// TIA Portal V15.1 export
// export: Created 2024-05-17T05:38:57.1842107Z, ExportSetting WithDefaults, DisplayName Totally Integrated Automation Portal, DisplayVersion V15.1 Update 5, DisplayName TIA Portal Openness, DisplayVersion V15.1 Update 5, DisplayName SINAMICS Startdrive Advanced, DisplayVersion V15.1, DisplayName G130, G150, S120, S150, SINAMICS MV, S210, DisplayVersion V15.1, DisplayName G110M, G120, G120C, G120D, G120P, DisplayVersion V15.1, DisplayName STEP 7 Professional, DisplayVersion V15.1 Update 5, DisplayName STEP 7 Safety, DisplayVersion V15.1, DisplayName WinCC Professional, DisplayVersion V15.1 Update 5, DisplayName SIMATIC Visualization Architect, DisplayVersion V15.1
FUNCTION "209210ZS01Passiv" : Void   // FC323, FBD
TITLE = 209210ZS01Passiv
{ S7_Optimized_Access := 'FALSE' }
AUTHOR : VCC
NAME : LocFunc
VERSION : 0.1
// stored: AutoNumber false, IsIECCheckEnabled false, SetENOAutomatically False, UDAEnableTagReadback false
   VAR_OUTPUT
      O_AlarmA : Bool;   // Alarm A
      O_AlarmB : Bool;   // Alarm B
      O_AlarmC : Bool;   // Alarm C
      O_AlarmD : Bool;   // Alarm D
      O_AlarmABCondition : Bool;   // Alarms resetable
      H_IAnim : Word;   // Icon Animation
   END_VAR
   VAR_TEMP
      TEMP0 : Bool;
   END_VAR
BEGIN

REGION Network 1: **** --------------------- ET200sp I/O --------------------- ****
END_REGION

REGION Network 2: **** 2.2 - Alarms - Alarm Generation **** 209000AK03JX36QF5240 - ET200sp I/O - Safety Card QF5240
   // Passivation alarm - ET200sp I/O - Safety Card QF5240
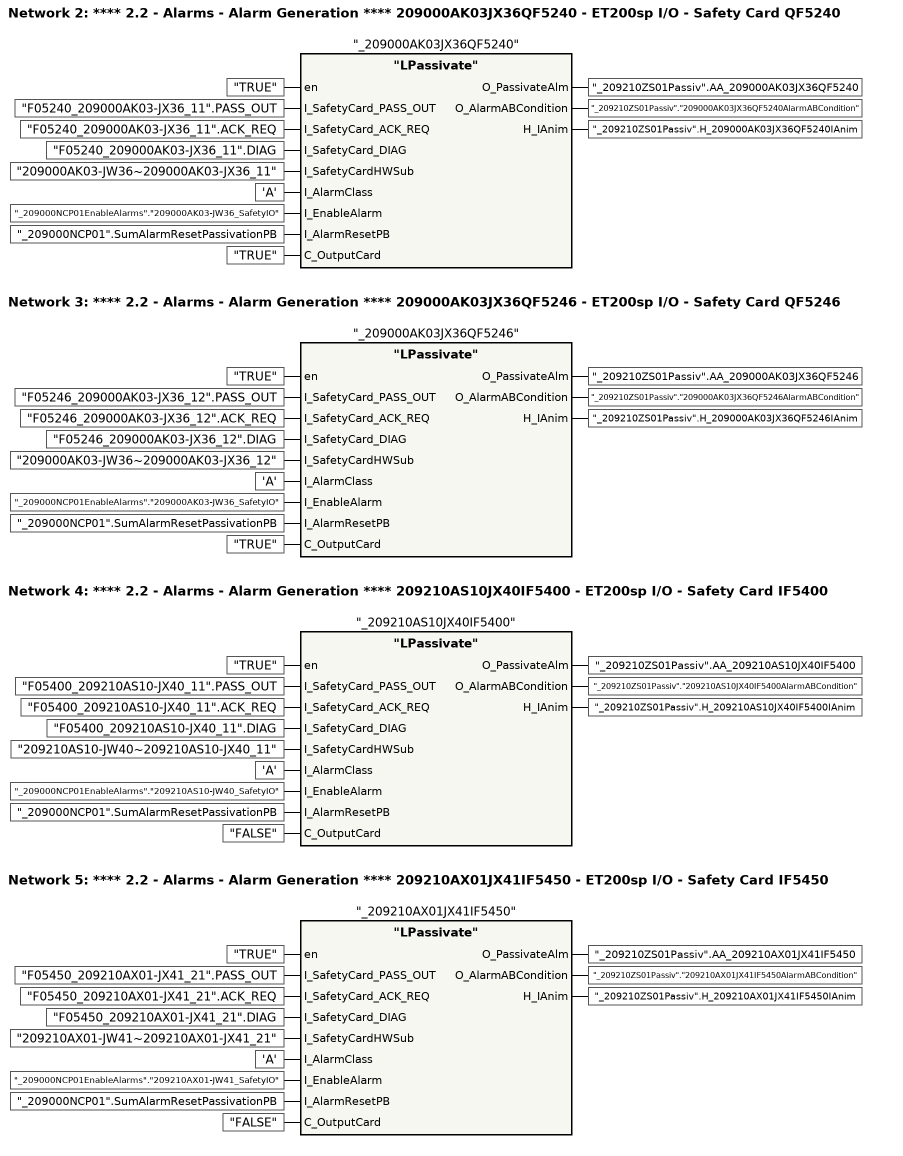
   IF "TRUE" THEN
       "_209000AK03JX36QF5240"(I_SafetyCard_PASS_OUT := "F05240_209000AK03-JX36_11".PASS_OUT,   // "LPassivate"
                               I_SafetyCard_ACK_REQ := "F05240_209000AK03-JX36_11".ACK_REQ,
                               I_SafetyCard_DIAG := "F05240_209000AK03-JX36_11".DIAG,
                               I_SafetyCardHWSub := "209000AK03-JW36~209000AK03-JX36_11",
                               I_AlarmClass := 'A',
                               I_EnableAlarm := "_209000NCP01EnableAlarms"."209000AK03-JW36_SafetyIO",
                               I_AlarmResetPB := "_209000NCP01".SumAlarmResetPassivationPB,
                               C_OutputCard := "TRUE",
                               O_PassivateAlm => "_209210ZS01Passiv".AA_209000AK03JX36QF5240,
                               O_AlarmABCondition => "_209210ZS01Passiv"."209000AK03JX36QF5240AlarmABCondition",
                               H_IAnim => "_209210ZS01Passiv".H_209000AK03JX36QF5240IAnim);
   END_IF;
END_REGION

REGION Network 3: **** 2.2 - Alarms - Alarm Generation **** 209000AK03JX36QF5246 - ET200sp I/O - Safety Card QF5246
   // Passivation alarm - ET200sp I/O - Safety Card QF5246
   IF "TRUE" THEN
       "_209000AK03JX36QF5246"(I_SafetyCard_PASS_OUT := "F05246_209000AK03-JX36_12".PASS_OUT,   // "LPassivate"
                               I_SafetyCard_ACK_REQ := "F05246_209000AK03-JX36_12".ACK_REQ,
                               I_SafetyCard_DIAG := "F05246_209000AK03-JX36_12".DIAG,
                               I_SafetyCardHWSub := "209000AK03-JW36~209000AK03-JX36_12",
                               I_AlarmClass := 'A',
                               I_EnableAlarm := "_209000NCP01EnableAlarms"."209000AK03-JW36_SafetyIO",
                               I_AlarmResetPB := "_209000NCP01".SumAlarmResetPassivationPB,
                               C_OutputCard := "TRUE",
                               O_PassivateAlm => "_209210ZS01Passiv".AA_209000AK03JX36QF5246,
                               O_AlarmABCondition => "_209210ZS01Passiv"."209000AK03JX36QF5246AlarmABCondition",
                               H_IAnim => "_209210ZS01Passiv".H_209000AK03JX36QF5246IAnim);
   END_IF;
END_REGION

REGION Network 4: **** 2.2 - Alarms - Alarm Generation **** 209210AS10JX40IF5400 - ET200sp I/O - Safety Card IF5400
   // Passivation alarm - ET200sp I/O - Safety Card IF5400
   IF "TRUE" THEN
       "_209210AS10JX40IF5400"(I_SafetyCard_PASS_OUT := "F05400_209210AS10-JX40_11".PASS_OUT,   // "LPassivate"
                               I_SafetyCard_ACK_REQ := "F05400_209210AS10-JX40_11".ACK_REQ,
                               I_SafetyCard_DIAG := "F05400_209210AS10-JX40_11".DIAG,
                               I_SafetyCardHWSub := "209210AS10-JW40~209210AS10-JX40_11",
                               I_AlarmClass := 'A',
                               I_EnableAlarm := "_209000NCP01EnableAlarms"."209210AS10-JW40_SafetyIO",
                               I_AlarmResetPB := "_209000NCP01".SumAlarmResetPassivationPB,
                               C_OutputCard := "FALSE",
                               O_PassivateAlm => "_209210ZS01Passiv".AA_209210AS10JX40IF5400,
                               O_AlarmABCondition => "_209210ZS01Passiv"."209210AS10JX40IF5400AlarmABCondition",
                               H_IAnim => "_209210ZS01Passiv".H_209210AS10JX40IF5400IAnim);
   END_IF;
END_REGION

REGION Network 5: **** 2.2 - Alarms - Alarm Generation **** 209210AX01JX41IF5450 - ET200sp I/O - Safety Card IF5450
   // Passivation alarm - ET200sp I/O - Safety Card IF5450
   IF "TRUE" THEN
       "_209210AX01JX41IF5450"(I_SafetyCard_PASS_OUT := "F05450_209210AX01-JX41_21".PASS_OUT,   // "LPassivate"
                               I_SafetyCard_ACK_REQ := "F05450_209210AX01-JX41_21".ACK_REQ,
                               I_SafetyCard_DIAG := "F05450_209210AX01-JX41_21".DIAG,
                               I_SafetyCardHWSub := "209210AX01-JW41~209210AX01-JX41_21",
                               I_AlarmClass := 'A',
                               I_EnableAlarm := "_209000NCP01EnableAlarms"."209210AX01-JW41_SafetyIO",
                               I_AlarmResetPB := "_209000NCP01".SumAlarmResetPassivationPB,
                               C_OutputCard := "FALSE",
                               O_PassivateAlm => "_209210ZS01Passiv".AA_209210AX01JX41IF5450,
                               O_AlarmABCondition => "_209210ZS01Passiv"."209210AX01JX41IF5450AlarmABCondition",
                               H_IAnim => "_209210ZS01Passiv".H_209210AX01JX41IF5450IAnim);
   END_IF;
END_REGION

REGION Network 6: **** 2.2 - Alarms - Alarm Generation **** 209210AS11JX42IF5500 - ET200sp I/O - Safety Card IF5500
   // Passivation alarm - ET200sp I/O - Safety Card IF5500
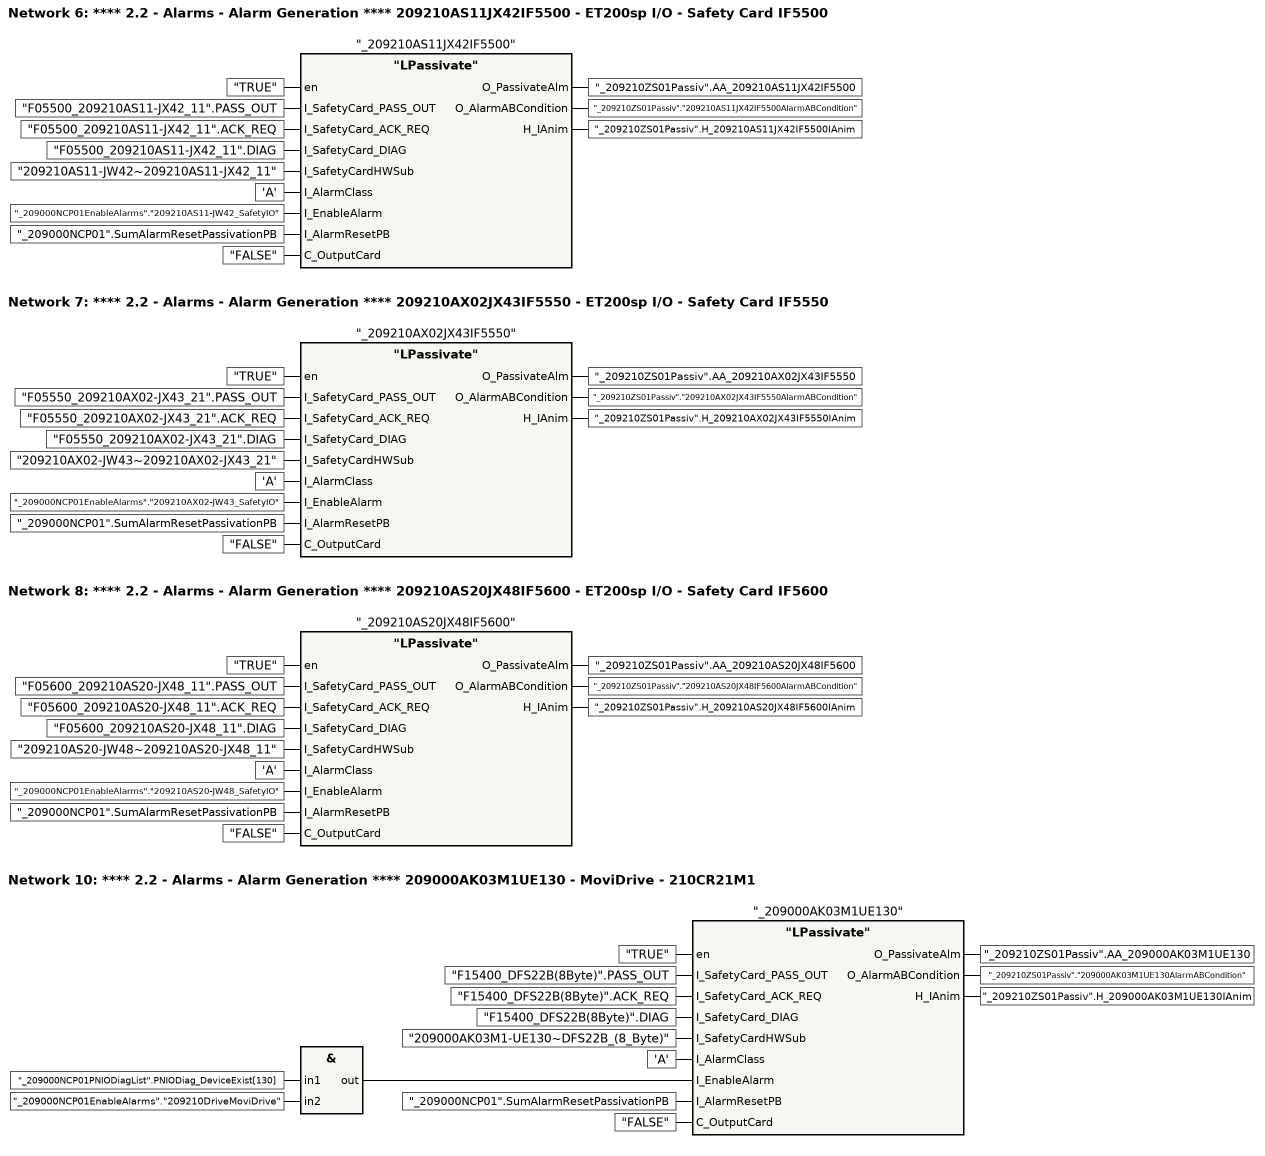
   IF "TRUE" THEN
       "_209210AS11JX42IF5500"(I_SafetyCard_PASS_OUT := "F05500_209210AS11-JX42_11".PASS_OUT,   // "LPassivate"
                               I_SafetyCard_ACK_REQ := "F05500_209210AS11-JX42_11".ACK_REQ,
                               I_SafetyCard_DIAG := "F05500_209210AS11-JX42_11".DIAG,
                               I_SafetyCardHWSub := "209210AS11-JW42~209210AS11-JX42_11",
                               I_AlarmClass := 'A',
                               I_EnableAlarm := "_209000NCP01EnableAlarms"."209210AS11-JW42_SafetyIO",
                               I_AlarmResetPB := "_209000NCP01".SumAlarmResetPassivationPB,
                               C_OutputCard := "FALSE",
                               O_PassivateAlm => "_209210ZS01Passiv".AA_209210AS11JX42IF5500,
                               O_AlarmABCondition => "_209210ZS01Passiv"."209210AS11JX42IF5500AlarmABCondition",
                               H_IAnim => "_209210ZS01Passiv".H_209210AS11JX42IF5500IAnim);
   END_IF;
END_REGION

REGION Network 7: **** 2.2 - Alarms - Alarm Generation **** 209210AX02JX43IF5550 - ET200sp I/O - Safety Card IF5550
   // Passivation alarm - ET200sp I/O - Safety Card IF5550
   IF "TRUE" THEN
       "_209210AX02JX43IF5550"(I_SafetyCard_PASS_OUT := "F05550_209210AX02-JX43_21".PASS_OUT,   // "LPassivate"
                               I_SafetyCard_ACK_REQ := "F05550_209210AX02-JX43_21".ACK_REQ,
                               I_SafetyCard_DIAG := "F05550_209210AX02-JX43_21".DIAG,
                               I_SafetyCardHWSub := "209210AX02-JW43~209210AX02-JX43_21",
                               I_AlarmClass := 'A',
                               I_EnableAlarm := "_209000NCP01EnableAlarms"."209210AX02-JW43_SafetyIO",
                               I_AlarmResetPB := "_209000NCP01".SumAlarmResetPassivationPB,
                               C_OutputCard := "FALSE",
                               O_PassivateAlm => "_209210ZS01Passiv".AA_209210AX02JX43IF5550,
                               O_AlarmABCondition => "_209210ZS01Passiv"."209210AX02JX43IF5550AlarmABCondition",
                               H_IAnim => "_209210ZS01Passiv".H_209210AX02JX43IF5550IAnim);
   END_IF;
END_REGION

REGION Network 8: **** 2.2 - Alarms - Alarm Generation **** 209210AS20JX48IF5600 - ET200sp I/O - Safety Card IF5600
   // Passivation alarm - ET200sp I/O - Safety Card IF5600
   IF "TRUE" THEN
       "_209210AS20JX48IF5600"(I_SafetyCard_PASS_OUT := "F05600_209210AS20-JX48_11".PASS_OUT,   // "LPassivate"
                               I_SafetyCard_ACK_REQ := "F05600_209210AS20-JX48_11".ACK_REQ,
                               I_SafetyCard_DIAG := "F05600_209210AS20-JX48_11".DIAG,
                               I_SafetyCardHWSub := "209210AS20-JW48~209210AS20-JX48_11",
                               I_AlarmClass := 'A',
                               I_EnableAlarm := "_209000NCP01EnableAlarms"."209210AS20-JW48_SafetyIO",
                               I_AlarmResetPB := "_209000NCP01".SumAlarmResetPassivationPB,
                               C_OutputCard := "FALSE",
                               O_PassivateAlm => "_209210ZS01Passiv".AA_209210AS20JX48IF5600,
                               O_AlarmABCondition => "_209210ZS01Passiv"."209210AS20JX48IF5600AlarmABCondition",
                               H_IAnim => "_209210ZS01Passiv".H_209210AS20JX48IF5600IAnim);
   END_IF;
END_REGION

REGION Network 9: **** --------------------- Drive --------------------- ****
END_REGION

REGION Network 10: **** 2.2 - Alarms - Alarm Generation **** 209000AK03M1UE130 - MoviDrive - 210CR21M1
   // Passivation alarm - MoviDrive - 210CR21M1
   IF "TRUE" THEN
       "_209000AK03M1UE130"(I_SafetyCard_PASS_OUT := "F15400_DFS22B(8Byte)".PASS_OUT,   // "LPassivate"
                            I_SafetyCard_ACK_REQ := "F15400_DFS22B(8Byte)".ACK_REQ,
                            I_SafetyCard_DIAG := "F15400_DFS22B(8Byte)".DIAG,
                            I_SafetyCardHWSub := "209000AK03M1-UE130~DFS22B_(8_Byte)",
                            I_AlarmClass := 'A',
                            I_EnableAlarm := "_209000NCP01PNIODiagList".PNIODiag_DeviceExist[130] AND "_209000NCP01EnableAlarms"."209210DriveMoviDrive",
                            I_AlarmResetPB := "_209000NCP01".SumAlarmResetPassivationPB,
                            C_OutputCard := "FALSE",
                            O_PassivateAlm => "_209210ZS01Passiv".AA_209000AK03M1UE130,
                            O_AlarmABCondition => "_209210ZS01Passiv"."209000AK03M1UE130AlarmABCondition",
                            H_IAnim => "_209210ZS01Passiv".H_209000AK03M1UE130IAnim);
   END_IF;
END_REGION

REGION Network 11: **** 2.2 - Alarms - Alarm Generation **** 209000AK03M4UE131 - MoviDrive - 210CS22M4ME1 (Power)
   // Passivation alarm - MoviDrive - 210CS22M4ME1 (Power)
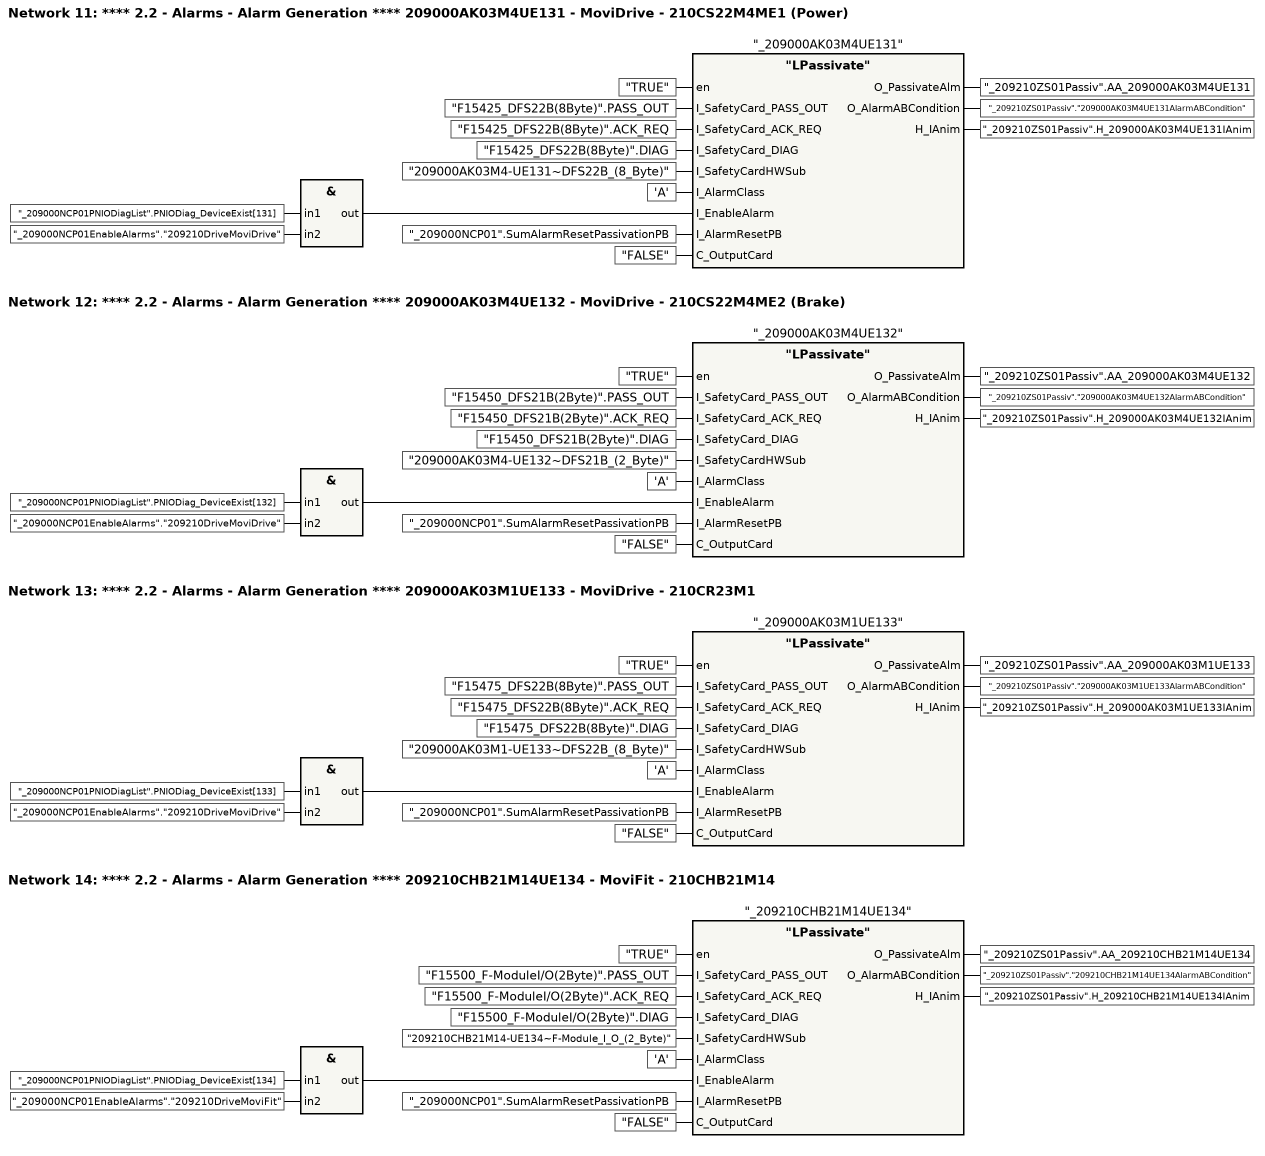
   IF "TRUE" THEN
       "_209000AK03M4UE131"(I_SafetyCard_PASS_OUT := "F15425_DFS22B(8Byte)".PASS_OUT,   // "LPassivate"
                            I_SafetyCard_ACK_REQ := "F15425_DFS22B(8Byte)".ACK_REQ,
                            I_SafetyCard_DIAG := "F15425_DFS22B(8Byte)".DIAG,
                            I_SafetyCardHWSub := "209000AK03M4-UE131~DFS22B_(8_Byte)",
                            I_AlarmClass := 'A',
                            I_EnableAlarm := "_209000NCP01PNIODiagList".PNIODiag_DeviceExist[131] AND "_209000NCP01EnableAlarms"."209210DriveMoviDrive",
                            I_AlarmResetPB := "_209000NCP01".SumAlarmResetPassivationPB,
                            C_OutputCard := "FALSE",
                            O_PassivateAlm => "_209210ZS01Passiv".AA_209000AK03M4UE131,
                            O_AlarmABCondition => "_209210ZS01Passiv"."209000AK03M4UE131AlarmABCondition",
                            H_IAnim => "_209210ZS01Passiv".H_209000AK03M4UE131IAnim);
   END_IF;
END_REGION

REGION Network 12: **** 2.2 - Alarms - Alarm Generation **** 209000AK03M4UE132 - MoviDrive - 210CS22M4ME2 (Brake)
   // Passivation alarm - MoviDrive - 210CS22M4ME2 (Brake)
   IF "TRUE" THEN
       "_209000AK03M4UE132"(I_SafetyCard_PASS_OUT := "F15450_DFS21B(2Byte)".PASS_OUT,   // "LPassivate"
                            I_SafetyCard_ACK_REQ := "F15450_DFS21B(2Byte)".ACK_REQ,
                            I_SafetyCard_DIAG := "F15450_DFS21B(2Byte)".DIAG,
                            I_SafetyCardHWSub := "209000AK03M4-UE132~DFS21B_(2_Byte)",
                            I_AlarmClass := 'A',
                            I_EnableAlarm := "_209000NCP01PNIODiagList".PNIODiag_DeviceExist[132] AND "_209000NCP01EnableAlarms"."209210DriveMoviDrive",
                            I_AlarmResetPB := "_209000NCP01".SumAlarmResetPassivationPB,
                            C_OutputCard := "FALSE",
                            O_PassivateAlm => "_209210ZS01Passiv".AA_209000AK03M4UE132,
                            O_AlarmABCondition => "_209210ZS01Passiv"."209000AK03M4UE132AlarmABCondition",
                            H_IAnim => "_209210ZS01Passiv".H_209000AK03M4UE132IAnim);
   END_IF;
END_REGION

REGION Network 13: **** 2.2 - Alarms - Alarm Generation **** 209000AK03M1UE133 - MoviDrive - 210CR23M1
   // Passivation alarm - MoviDrive - 210CR23M1
   IF "TRUE" THEN
       "_209000AK03M1UE133"(I_SafetyCard_PASS_OUT := "F15475_DFS22B(8Byte)".PASS_OUT,   // "LPassivate"
                            I_SafetyCard_ACK_REQ := "F15475_DFS22B(8Byte)".ACK_REQ,
                            I_SafetyCard_DIAG := "F15475_DFS22B(8Byte)".DIAG,
                            I_SafetyCardHWSub := "209000AK03M1-UE133~DFS22B_(8_Byte)",
                            I_AlarmClass := 'A',
                            I_EnableAlarm := "_209000NCP01PNIODiagList".PNIODiag_DeviceExist[133] AND "_209000NCP01EnableAlarms"."209210DriveMoviDrive",
                            I_AlarmResetPB := "_209000NCP01".SumAlarmResetPassivationPB,
                            C_OutputCard := "FALSE",
                            O_PassivateAlm => "_209210ZS01Passiv".AA_209000AK03M1UE133,
                            O_AlarmABCondition => "_209210ZS01Passiv"."209000AK03M1UE133AlarmABCondition",
                            H_IAnim => "_209210ZS01Passiv".H_209000AK03M1UE133IAnim);
   END_IF;
END_REGION

REGION Network 14: **** 2.2 - Alarms - Alarm Generation **** 209210CHB21M14UE134 - MoviFit - 210CHB21M14
   // Passivation alarm - MoviFit - 210CHB21M14
   IF "TRUE" THEN
       "_209210CHB21M14UE134"(I_SafetyCard_PASS_OUT := "F15500_F-ModuleI/O(2Byte)".PASS_OUT,   // "LPassivate"
                              I_SafetyCard_ACK_REQ := "F15500_F-ModuleI/O(2Byte)".ACK_REQ,
                              I_SafetyCard_DIAG := "F15500_F-ModuleI/O(2Byte)".DIAG,
                              I_SafetyCardHWSub := "209210CHB21M14-UE134~F-Module_I_O_(2_Byte)",
                              I_AlarmClass := 'A',
                              I_EnableAlarm := "_209000NCP01PNIODiagList".PNIODiag_DeviceExist[134] AND "_209000NCP01EnableAlarms"."209210DriveMoviFit",
                              I_AlarmResetPB := "_209000NCP01".SumAlarmResetPassivationPB,
                              C_OutputCard := "FALSE",
                              O_PassivateAlm => "_209210ZS01Passiv".AA_209210CHB21M14UE134,
                              O_AlarmABCondition => "_209210ZS01Passiv"."209210CHB21M14UE134AlarmABCondition",
                              H_IAnim => "_209210ZS01Passiv".H_209210CHB21M14UE134IAnim);
   END_IF;
END_REGION

REGION Network 15: **** -------------------------------------------------- ****
END_REGION

REGION Network 16: **** 4.6 - Machine Status - Indications **** Icon animation
   // Icon animation
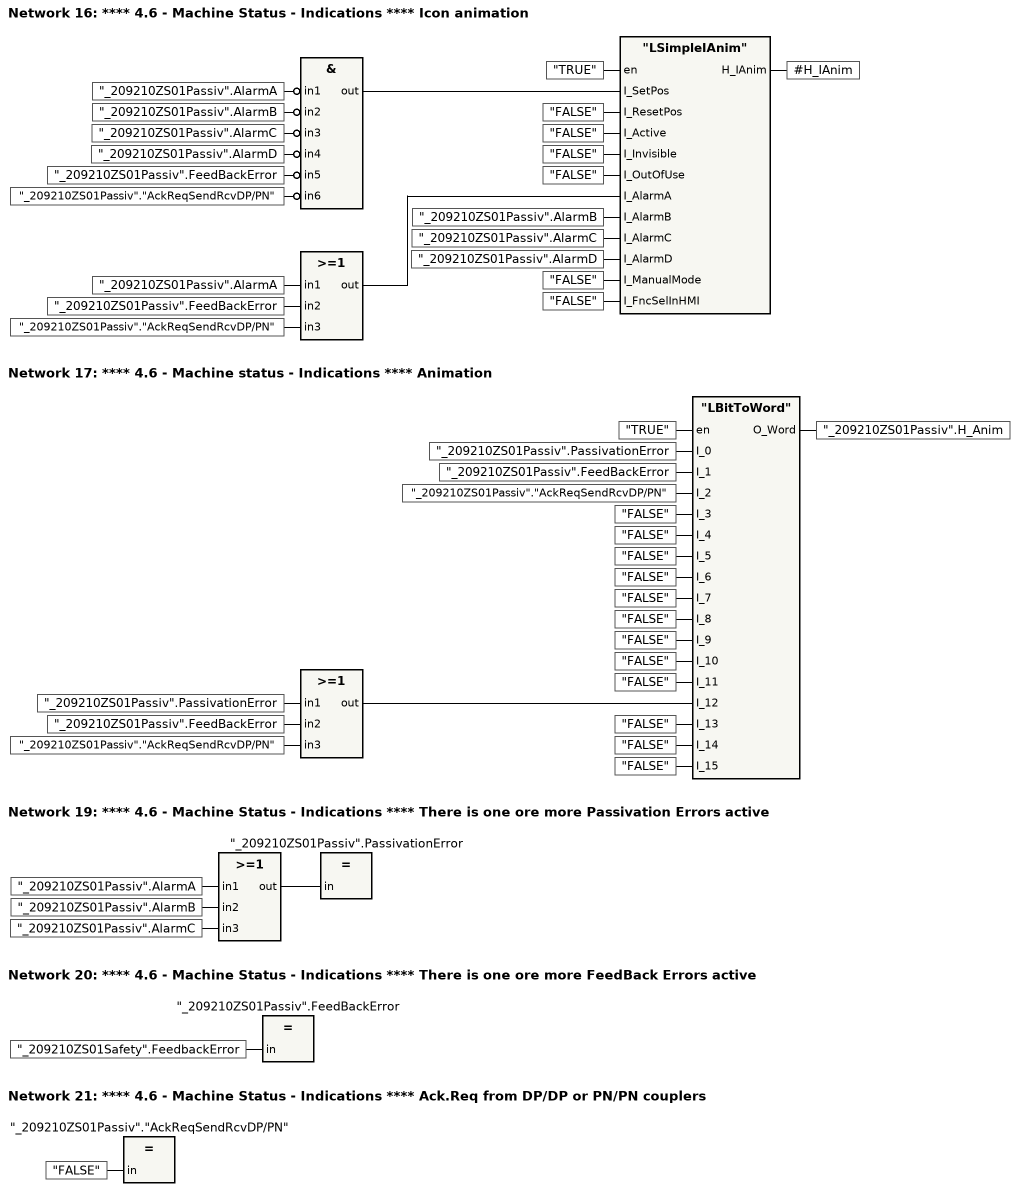
   IF "TRUE" THEN
       "LSimpleIAnim"(I_SetPos := NOT "_209210ZS01Passiv".AlarmA AND NOT "_209210ZS01Passiv".AlarmB AND NOT "_209210ZS01Passiv".AlarmC AND NOT "_209210ZS01Passiv".AlarmD AND NOT "_209210ZS01Passiv".FeedBackError AND NOT "_209210ZS01Passiv"."AckReqSendRcvDP/PN",
                      I_ResetPos := "FALSE",
                      I_Active := "FALSE",
                      I_Invisible := "FALSE",
                      I_OutOfUse := "FALSE",
                      I_AlarmA := "_209210ZS01Passiv".AlarmA OR "_209210ZS01Passiv".FeedBackError OR "_209210ZS01Passiv"."AckReqSendRcvDP/PN",
                      I_AlarmB := "_209210ZS01Passiv".AlarmB,
                      I_AlarmC := "_209210ZS01Passiv".AlarmC,
                      I_AlarmD := "_209210ZS01Passiv".AlarmD,
                      I_ManualMode := "FALSE",
                      I_FncSelInHMI := "FALSE",
                      H_IAnim => #H_IAnim);
   END_IF;
END_REGION

REGION Network 17: **** 4.6 - Machine status - Indications **** Animation
   // Animation
   IF "TRUE" THEN
       "LBitToWord"(I_0 := "_209210ZS01Passiv".PassivationError,
                    I_1 := "_209210ZS01Passiv".FeedBackError,
                    I_2 := "_209210ZS01Passiv"."AckReqSendRcvDP/PN",
                    I_3 := "FALSE",
                    I_4 := "FALSE",
                    I_5 := "FALSE",
                    I_6 := "FALSE",
                    I_7 := "FALSE",
                    I_8 := "FALSE",
                    I_9 := "FALSE",
                    I_10 := "FALSE",
                    I_11 := "FALSE",
                    I_12 := "_209210ZS01Passiv".PassivationError OR "_209210ZS01Passiv".FeedBackError OR "_209210ZS01Passiv"."AckReqSendRcvDP/PN",
                    I_13 := "FALSE",
                    I_14 := "FALSE",
                    I_15 := "FALSE",
                    O_Word => "_209210ZS01Passiv".H_Anim);
   END_IF;
END_REGION

NETWORK
TITLE = **** 4.6 - Machine Status - Indications **** Animation DB number
// DB number
      OPN   "_209210ZS01Passiv";
      L     DBNO;
      T     "_209210ZS01Passiv".H_DBnr;

REGION Network 19: **** 4.6 - Machine Status - Indications **** There is one ore more Passivation Errors active
   // There is one ore more Passivation Errors active
   "_209210ZS01Passiv".PassivationError := "_209210ZS01Passiv".AlarmA OR "_209210ZS01Passiv".AlarmB OR "_209210ZS01Passiv".AlarmC;
END_REGION

REGION Network 20: **** 4.6 - Machine Status - Indications **** There is one ore more FeedBack Errors active
   // There is one ore more FeedBack Errors active
   "_209210ZS01Passiv".FeedBackError := "_209210ZS01Safety".FeedbackError;
END_REGION

REGION Network 21: **** 4.6 - Machine Status - Indications **** Ack.Req from DP/DP or PN/PN couplers
   // Ack.Req from DP/DP or PN/PN couplers
   "_209210ZS01Passiv"."AckReqSendRcvDP/PN" := "FALSE";
END_REGION

REGION Network 22: **** 9 - Alarm Summary **** Alarm AB Condition
   // Alarm AB condition
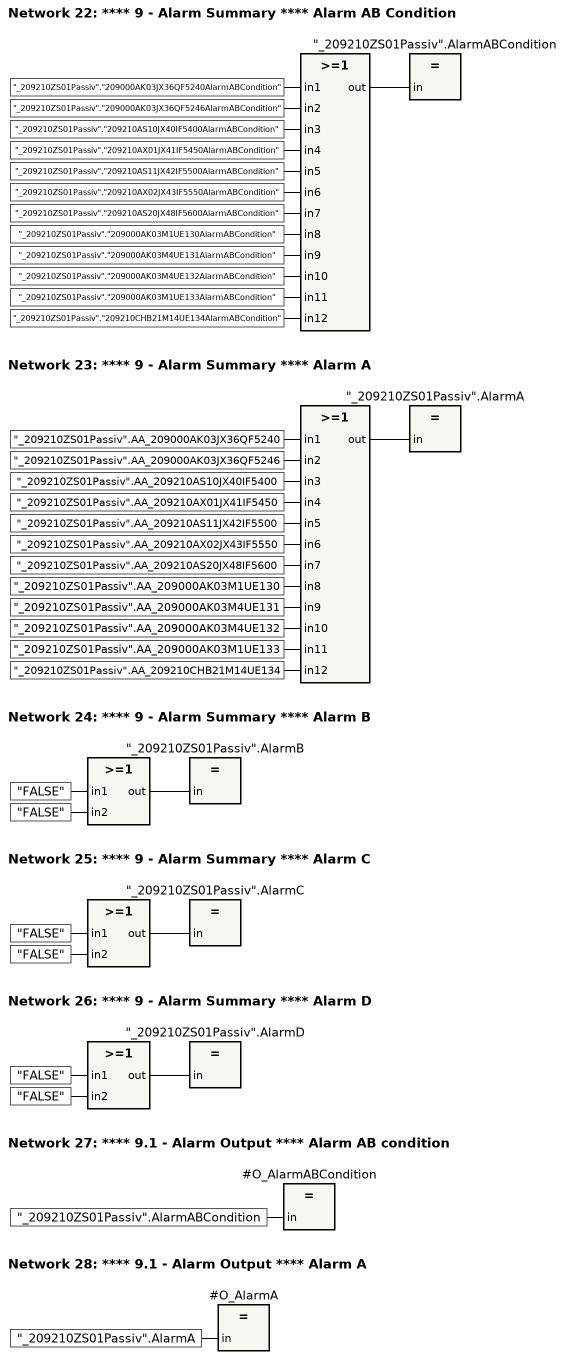
   "_209210ZS01Passiv".AlarmABCondition := "_209210ZS01Passiv"."209000AK03JX36QF5240AlarmABCondition" OR "_209210ZS01Passiv"."209000AK03JX36QF5246AlarmABCondition" OR "_209210ZS01Passiv"."209210AS10JX40IF5400AlarmABCondition" OR "_209210ZS01Passiv"."209210AX01JX41IF5450AlarmABCondition" OR "_209210ZS01Passiv"."209210AS11JX42IF5500AlarmABCondition" OR "_209210ZS01Passiv"."209210AX02JX43IF5550AlarmABCondition" OR "_209210ZS01Passiv"."209210AS20JX48IF5600AlarmABCondition" OR "_209210ZS01Passiv"."209000AK03M1UE130AlarmABCondition" OR "_209210ZS01Passiv"."209000AK03M4UE131AlarmABCondition" OR "_209210ZS01Passiv"."209000AK03M4UE132AlarmABCondition" OR "_209210ZS01Passiv"."209000AK03M1UE133AlarmABCondition" OR "_209210ZS01Passiv"."209210CHB21M14UE134AlarmABCondition";
END_REGION

REGION Network 23: **** 9 - Alarm Summary **** Alarm A
   // Summary of alarms A
   "_209210ZS01Passiv".AlarmA := "_209210ZS01Passiv".AA_209000AK03JX36QF5240 OR "_209210ZS01Passiv".AA_209000AK03JX36QF5246 OR "_209210ZS01Passiv".AA_209210AS10JX40IF5400 OR "_209210ZS01Passiv".AA_209210AX01JX41IF5450 OR "_209210ZS01Passiv".AA_209210AS11JX42IF5500 OR "_209210ZS01Passiv".AA_209210AX02JX43IF5550 OR "_209210ZS01Passiv".AA_209210AS20JX48IF5600 OR "_209210ZS01Passiv".AA_209000AK03M1UE130 OR "_209210ZS01Passiv".AA_209000AK03M4UE131 OR "_209210ZS01Passiv".AA_209000AK03M4UE132 OR "_209210ZS01Passiv".AA_209000AK03M1UE133 OR "_209210ZS01Passiv".AA_209210CHB21M14UE134;
END_REGION

REGION Network 24: **** 9 - Alarm Summary **** Alarm B
   // Summary of alarms B
   "_209210ZS01Passiv".AlarmB := "FALSE" OR "FALSE";
END_REGION

REGION Network 25: **** 9 - Alarm Summary **** Alarm C
   // Summary of alarms C
   "_209210ZS01Passiv".AlarmC := "FALSE" OR "FALSE";
END_REGION

REGION Network 26: **** 9 - Alarm Summary **** Alarm D
   // Summary of alarms D
   "_209210ZS01Passiv".AlarmD := "FALSE" OR "FALSE";
END_REGION

REGION Network 27: **** 9.1 - Alarm Output **** Alarm AB condition
   // Alarm AB condition
   #O_AlarmABCondition := "_209210ZS01Passiv".AlarmABCondition;
END_REGION

REGION Network 28: **** 9.1 - Alarm Output **** Alarm A
   // Output Alarm A
   #O_AlarmA := "_209210ZS01Passiv".AlarmA;
END_REGION

REGION Network 29: **** 9.1 - Alarm Output **** Alarm B
   // Output Alarm B
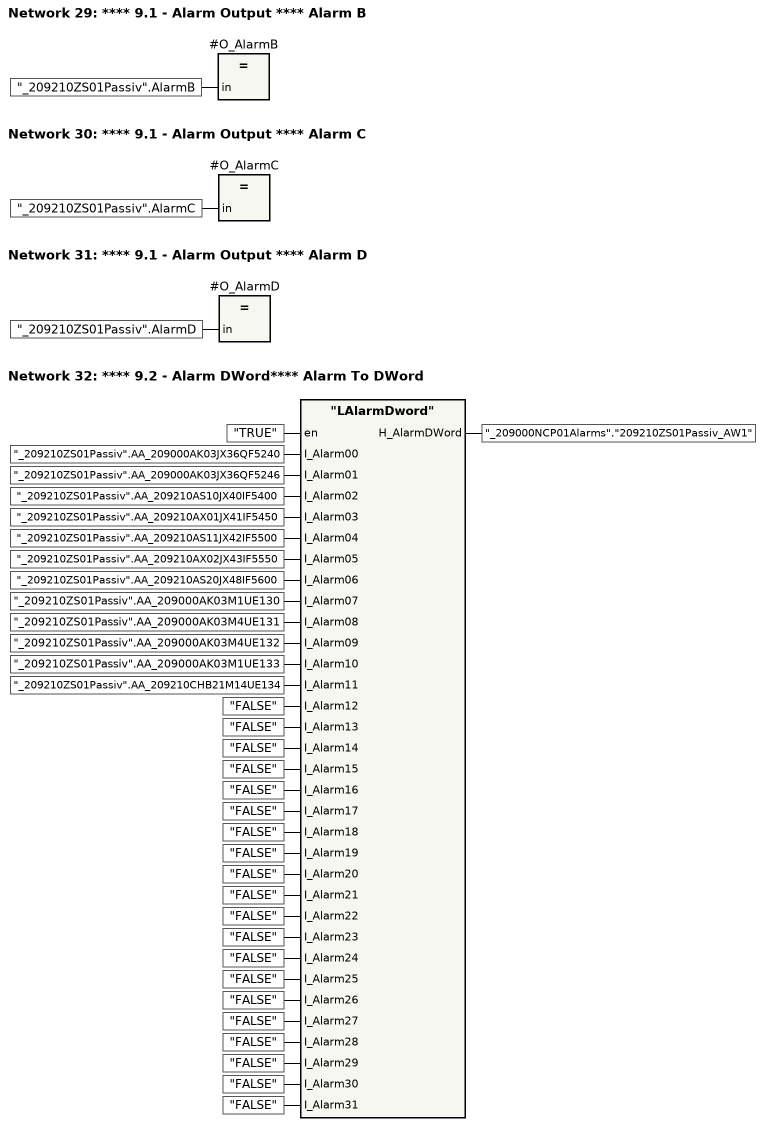
   #O_AlarmB := "_209210ZS01Passiv".AlarmB;
END_REGION

REGION Network 30: **** 9.1 - Alarm Output **** Alarm C
   // Output Alarm C
   #O_AlarmC := "_209210ZS01Passiv".AlarmC;
END_REGION

REGION Network 31: **** 9.1 - Alarm Output **** Alarm D
   // Output Alarm D
   #O_AlarmD := "_209210ZS01Passiv".AlarmD;
END_REGION

REGION Network 32: **** 9.2 - Alarm DWord**** Alarm To DWord
   // Alarm Word
   IF "TRUE" THEN
       "LAlarmDword"(I_Alarm00 := "_209210ZS01Passiv".AA_209000AK03JX36QF5240,
                     I_Alarm01 := "_209210ZS01Passiv".AA_209000AK03JX36QF5246,
                     I_Alarm02 := "_209210ZS01Passiv".AA_209210AS10JX40IF5400,
                     I_Alarm03 := "_209210ZS01Passiv".AA_209210AX01JX41IF5450,
                     I_Alarm04 := "_209210ZS01Passiv".AA_209210AS11JX42IF5500,
                     I_Alarm05 := "_209210ZS01Passiv".AA_209210AX02JX43IF5550,
                     I_Alarm06 := "_209210ZS01Passiv".AA_209210AS20JX48IF5600,
                     I_Alarm07 := "_209210ZS01Passiv".AA_209000AK03M1UE130,
                     I_Alarm08 := "_209210ZS01Passiv".AA_209000AK03M4UE131,
                     I_Alarm09 := "_209210ZS01Passiv".AA_209000AK03M4UE132,
                     I_Alarm10 := "_209210ZS01Passiv".AA_209000AK03M1UE133,
                     I_Alarm11 := "_209210ZS01Passiv".AA_209210CHB21M14UE134,
                     I_Alarm12 := "FALSE",
                     I_Alarm13 := "FALSE",
                     I_Alarm14 := "FALSE",
                     I_Alarm15 := "FALSE",
                     I_Alarm16 := "FALSE",
                     I_Alarm17 := "FALSE",
                     I_Alarm18 := "FALSE",
                     I_Alarm19 := "FALSE",
                     I_Alarm20 := "FALSE",
                     I_Alarm21 := "FALSE",
                     I_Alarm22 := "FALSE",
                     I_Alarm23 := "FALSE",
                     I_Alarm24 := "FALSE",
                     I_Alarm25 := "FALSE",
                     I_Alarm26 := "FALSE",
                     I_Alarm27 := "FALSE",
                     I_Alarm28 := "FALSE",
                     I_Alarm29 := "FALSE",
                     I_Alarm30 := "FALSE",
                     I_Alarm31 := "FALSE",
                     H_AlarmDWord => "_209000NCP01Alarms"."209210ZS01Passiv_AW1");
   END_IF;
END_REGION
END_FUNCTION
